SYSTEM Waterfilter
  (* Version 1.0, 2023-01-19, AK124017 *)
  APPLICATION Application
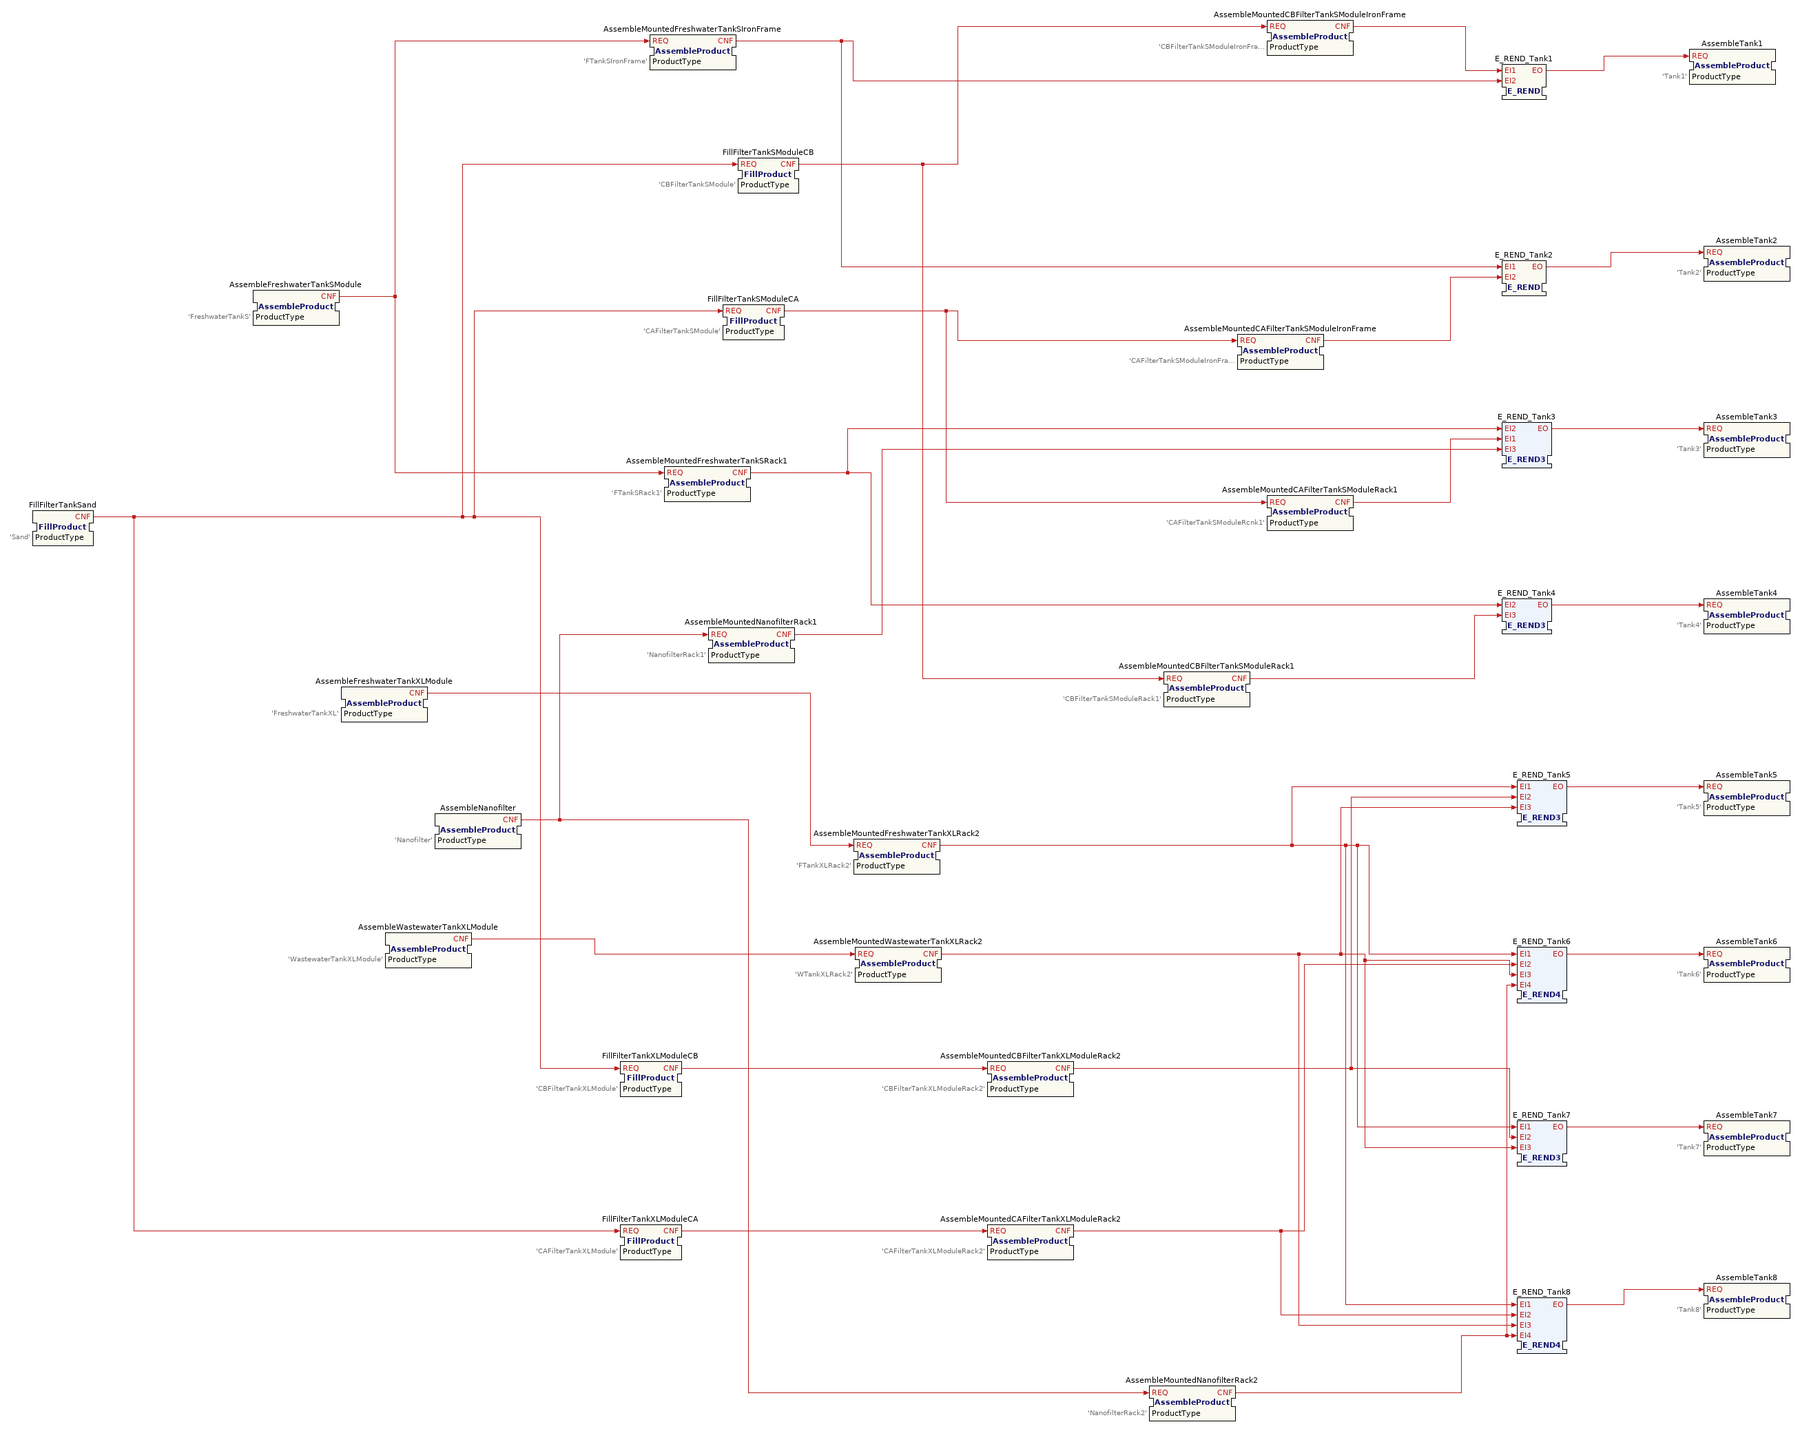
    FBS
      AssembleTank1 : AssembleProduct(ProductType := 'Tank1');
      AssembleTank2 : AssembleProduct(ProductType := 'Tank2');
      AssembleTank3 : AssembleProduct(ProductType := 'Tank3');
      AssembleTank4 : AssembleProduct(ProductType := 'Tank4');
      AssembleTank5 : AssembleProduct(ProductType := 'Tank5');
      AssembleTank6 : AssembleProduct(ProductType := 'Tank6');
      AssembleTank7 : AssembleProduct(ProductType := 'Tank7');
      AssembleTank8 : AssembleProduct(ProductType := 'Tank8');
      E_REND_Tank2 : E_REND;
      E_REND_Tank1 : E_REND;
      AssembleMountedFreshwaterTankSIronFrame : AssembleProduct(ProductType := 'FTankSIronFrame');
      AssembleMountedCBFilterTankSModuleIronFrame : AssembleProduct(ProductType := 'CBFilterTankSModuleIronFrame');
      AssembleMountedCAFilterTankSModuleIronFrame : AssembleProduct(ProductType := 'CAFilterTankSModuleIronFrame');
      AssembleMountedFreshwaterTankSRack1 : AssembleProduct(ProductType := 'FTankSRack1');
      AssembleMountedCAFilterTankSModuleRack1 : AssembleProduct(ProductType := 'CAFilterTankSModuleRcnk1');
      AssembleMountedCBFilterTankSModuleRack1 : AssembleProduct(ProductType := 'CBFilterTankSModuleRack1');
      AssembleMountedNanofilterRack1 : AssembleProduct(ProductType := 'NanofilterRack1');
      AssembleMountedFreshwaterTankXLRack2 : AssembleProduct(ProductType := 'FTankXLRack2');
      AssembleMountedCBFilterTankXLModuleRack2 : AssembleProduct(ProductType := 'CBFilterTankXLModuleRack2');
      AssembleMountedCAFilterTankXLModuleRack2 : AssembleProduct(ProductType := 'CAFilterTankXLModuleRack2');
      AssembleMountedWastewaterTankXLRack2 : AssembleProduct(ProductType := 'WTankXLRack2');
      AssembleMountedNanofilterRack2 : AssembleProduct(ProductType := 'NanofilterRack2');
      FillFilterTankSModuleCB : FillProduct(ProductType := 'CBFilterTankSModule');
      FillFilterTankSModuleCA : FillProduct(ProductType := 'CAFilterTankSModule');
      FillFilterTankXLModuleCA : FillProduct(ProductType := 'CAFilterTankXLModule');
      FillFilterTankXLModuleCB : FillProduct(ProductType := 'CBFilterTankXLModule');
      AssembleNanofilter : AssembleProduct(ProductType := 'Nanofilter');
      AssembleWastewaterTankXLModule : AssembleProduct(ProductType := 'WastewaterTankXLModule');
      AssembleFreshwaterTankXLModule : AssembleProduct(ProductType := 'FreshwaterTankXL');
      AssembleFreshwaterTankSModule : AssembleProduct(ProductType := 'FreshwaterTankS');
      FillFilterTankSand : FillProduct(ProductType := 'Sand');
    END_FBS
    SUBAPPS
      E_REND_Tank8 : E_REND4;
      E_REND_Tank7 : E_REND3;
      E_REND_Tank6 : E_REND4;
      E_REND_Tank5 : E_REND3;
      E_REND_Tank4 : E_REND3;
      E_REND_Tank3 : E_REND3;
    END_SUBAPPS
    EVENT_CONNECTIONS
      E_REND_Tank8.EO TO AssembleTank8.REQ;
      E_REND_Tank7.EO TO AssembleTank7.REQ;
      E_REND_Tank6.EO TO AssembleTank6.REQ;
      E_REND_Tank3.EO TO AssembleTank3.REQ;
      E_REND_Tank4.EO TO AssembleTank4.REQ;
      E_REND_Tank5.EO TO AssembleTank5.REQ;
      E_REND_Tank2.EO TO AssembleTank2.REQ;
      E_REND_Tank1.EO TO AssembleTank1.REQ;
      AssembleMountedCBFilterTankSModuleIronFrame.CNF TO E_REND_Tank1.EI1;
      AssembleMountedFreshwaterTankSIronFrame.CNF TO E_REND_Tank1.EI2;
      AssembleMountedFreshwaterTankSIronFrame.CNF TO E_REND_Tank2.EI1;
      AssembleMountedCAFilterTankSModuleIronFrame.CNF TO E_REND_Tank2.EI2;
      AssembleMountedFreshwaterTankSRack1.CNF TO E_REND_Tank3.EI2;
      AssembleMountedFreshwaterTankSRack1.CNF TO E_REND_Tank4.EI2;
      AssembleMountedCAFilterTankSModuleRack1.CNF TO E_REND_Tank3.EI1;
      AssembleMountedCBFilterTankSModuleRack1.CNF TO E_REND_Tank4.EI3;
      AssembleMountedNanofilterRack1.CNF TO E_REND_Tank3.EI3;
      AssembleMountedFreshwaterTankXLRack2.CNF TO E_REND_Tank5.EI1;
      AssembleMountedFreshwaterTankXLRack2.CNF TO E_REND_Tank6.EI1;
      AssembleMountedFreshwaterTankXLRack2.CNF TO E_REND_Tank7.EI1;
      AssembleMountedFreshwaterTankXLRack2.CNF TO E_REND_Tank8.EI1;
      AssembleMountedCBFilterTankXLModuleRack2.CNF TO E_REND_Tank5.EI2;
      AssembleMountedCBFilterTankXLModuleRack2.CNF TO E_REND_Tank7.EI2;
      AssembleMountedCAFilterTankXLModuleRack2.CNF TO E_REND_Tank8.EI2;
      AssembleMountedCAFilterTankXLModuleRack2.CNF TO E_REND_Tank6.EI2;
      AssembleMountedWastewaterTankXLRack2.CNF TO E_REND_Tank5.EI3;
      AssembleMountedWastewaterTankXLRack2.CNF TO E_REND_Tank6.EI3;
      AssembleMountedWastewaterTankXLRack2.CNF TO E_REND_Tank7.EI3;
      AssembleMountedWastewaterTankXLRack2.CNF TO E_REND_Tank8.EI3;
      AssembleMountedNanofilterRack2.CNF TO E_REND_Tank8.EI4;
      AssembleMountedNanofilterRack2.CNF TO E_REND_Tank6.EI4;
      FillFilterTankSModuleCB.CNF TO AssembleMountedCBFilterTankSModuleIronFrame.REQ;
      FillFilterTankSModuleCA.CNF TO AssembleMountedCAFilterTankSModuleIronFrame.REQ;
      FillFilterTankSModuleCA.CNF TO AssembleMountedCAFilterTankSModuleRack1.REQ;
      FillFilterTankSModuleCB.CNF TO AssembleMountedCBFilterTankSModuleRack1.REQ;
      FillFilterTankXLModuleCB.CNF TO AssembleMountedCBFilterTankXLModuleRack2.REQ;
      FillFilterTankXLModuleCA.CNF TO AssembleMountedCAFilterTankXLModuleRack2.REQ;
      AssembleNanofilter.CNF TO AssembleMountedNanofilterRack1.REQ;
      AssembleNanofilter.CNF TO AssembleMountedNanofilterRack2.REQ;
      AssembleWastewaterTankXLModule.CNF TO AssembleMountedWastewaterTankXLRack2.REQ;
      AssembleFreshwaterTankXLModule.CNF TO AssembleMountedFreshwaterTankXLRack2.REQ;
      AssembleFreshwaterTankSModule.CNF TO AssembleMountedFreshwaterTankSIronFrame.REQ;
      AssembleFreshwaterTankSModule.CNF TO AssembleMountedFreshwaterTankSRack1.REQ;
      FillFilterTankSand.CNF TO FillFilterTankSModuleCB.REQ;
      FillFilterTankSand.CNF TO FillFilterTankSModuleCA.REQ;
      FillFilterTankSand.CNF TO FillFilterTankXLModuleCB.REQ;
      FillFilterTankSand.CNF TO FillFilterTankXLModuleCA.REQ;
    END_CONNECTIONS
  END_APPLICATION
END_SYSTEM
